// TIA Portal V19 export
FUNCTION_BLOCK "TYPIC_C104_IF_NSI"   // FB91, FBD
TITLE = TYPIC_C104_IF_NSI: Noodstroominstallatie
{ S7_Optimized_Access := 'TRUE' }
AUTHOR : OCOTECH
FAMILY : Typical
NAME : C104.701
// Logisch Object Besturing: C104.701
// 
// De interne functie Noodstroominstallatie verzorgt de bewaking van de noodstroominstallatie.
// stored: MemoryReserve 10, SetENOAutomatically false
   VAR_INPUT
      IN_NSI_BSC1 { ExternalAccessible := 'False'; ExternalVisible := 'False'; ExternalWritable := 'False'} : Bool;   // Noodstroominstallatie beschikbaar
      IN_NSI_BSC2 { ExternalAccessible := 'False'; ExternalVisible := 'False'; ExternalWritable := 'False'} : Bool;   // Noodstroominstallatie niet beschikbaar
      IN_NSI_BSC3 { ExternalAccessible := 'False'; ExternalVisible := 'False'; ExternalWritable := 'False'} : Bool;   // Noodstroominstallatie beperkt beschikbaar
      IN_NSI_ENE_TOT { ExternalAccessible := 'False'; ExternalVisible := 'False'; ExternalWritable := 'False'} : Real;   // Totaal energieverbruik noodstroominstallatie
      IN_AUT_C104 { ExternalAccessible := 'False'; ExternalVisible := 'False'; ExternalWritable := 'False'} : Bool;   // Beveiligingen: serie geschakelde terugmelding (1 = OK)
   END_VAR
   VAR_OUTPUT
      VAR_IF_NSI { ExternalAccessible := 'False'; ExternalVisible := 'False'; ExternalWritable := 'False'} : "C104_VAR_IF_NSI_TYPIC";   // Struct met alle variabelen naar bovenliggende functies
   END_VAR
   VAR
      VAR { ExternalWritable := 'False'} : Struct   // Variabelen
         BSC1 { ExternalAccessible := 'False'; ExternalVisible := 'False'} : Bool;   // Noodstroominstallatie beschikbaar
         BSC2 { ExternalAccessible := 'False'; ExternalVisible := 'False'} : Bool;   // Noodstroominstallatie niet beschikbaar
         BSC3 { ExternalAccessible := 'False'; ExternalVisible := 'False'} : Bool;   // Noodstroominstallatie beperkt beschikbaar
         ENE_TOT { ExternalAccessible := 'False'; ExternalVisible := 'False'} : Real;   // Totaal energieverbruik noodstroominstallatie
      END_STRUCT;
   END_VAR
BEGIN

REGION Network 1: START
END_REGION

REGION Network 2: +++ Verwerking meetwaarden en statussen +++
   // De meetwaarden en statussen van de noodstroominstallatie worden ontvangen vanuit de interne sturing.
END_REGION

REGION Network 3: +++ Storingen +++
   // Verwerken van de storingsmeldingen (inputs).
END_REGION

REGION Network 4 (SCL): EINDE
   // Variabelen van intern scada rakvlak naar outputs copieren
   #VAR_IF_NSI.BSC1 := #VAR.BSC1;
   #VAR_IF_NSI.BSC2 := #VAR.BSC2;
   #VAR_IF_NSI.BSC3 := #VAR.BSC3;
   #VAR_IF_NSI.ENE_TOT := #VAR.ENE_TOT;
END_REGION
END_FUNCTION_BLOCK
